// TIA Portal V19 export
TYPE "UDT_AINFAULTS"
   STRUCT
      ctrl : Struct   // External data (Primary fault data - alarm & plc ackn)
         alarm_hh : Bool := false;
         alarm_ll : Bool := false;
         bit10 : Bool := false;
         bit11 : Bool := false;
         bit12 : Bool := false;
         bit13 : Bool := false;
         bit14 : Bool := false;
         bit15 : Bool := false;
         plcackn_hh : Bool := false;
         plcackn_ll : Bool := false;
         bit2 : Bool := false;
         bit3 : Bool := false;
         bit4 : Bool := false;
         bit5 : Bool := false;
         bit6 : Bool := false;
         bit7 : Bool := false;
      END_STRUCT;
      status : Struct   // External data (Secondary fault data - siren & hmi ackn)
         siren_hh : Bool := false;
         siren_ll : Bool := false;
         bit10 : Bool := false;
         bit11 : Bool := false;
         bit12 : Bool := false;
         bit13 : Bool := false;
         bit14 : Bool := false;
         bit15 : Bool := false;
         hmiackn_hh : Bool := false;
         hmiackn_ll : Bool := false;
         bit2 : Bool := false;
         bit3 : Bool := false;
         bit4 : Bool := false;
         bit5 : Bool := false;
         bit6 : Bool := false;
         bit7 : Bool := false;
      END_STRUCT;
   END_STRUCT;
END_TYPE
